TYPE ST_TestStruct :
STRUCT
	nIndex: UDINT;
	aData : ARRAY[1..1020] OF BYTE;
END_STRUCT
END_TYPE

(* stored: Version 1.1.0.1
   DUT ST_TestStruct: Id {8e4b7aa3-a05a-427b-a09b-7949583c16b7} *)
